FUNCTION_BLOCK FB_System_MVKW_Ablaufsteuerung
VAR_IN_OUT
	Zustand					: ST_System_MVKW_Zustand;
	Stellwert				: ST_System_MVKW_Stellwert;
	Steuerung				: ST_System_MVKW_Steuerung;
END_VAR
VAR_INPUT
	Zustand_Stellventil		: ST_SV_Zustand;
	Zustand_Pumpe			: ST_PU_Zustand;
END_VAR
VAR_OUTPUT
END_VAR
VAR
	E_System_DLK_Zustand_Status_Stoerung	: SINT;
	E_System_DLK_Zustand_Status_Idle_Sperre	: SINT;
END_VAR

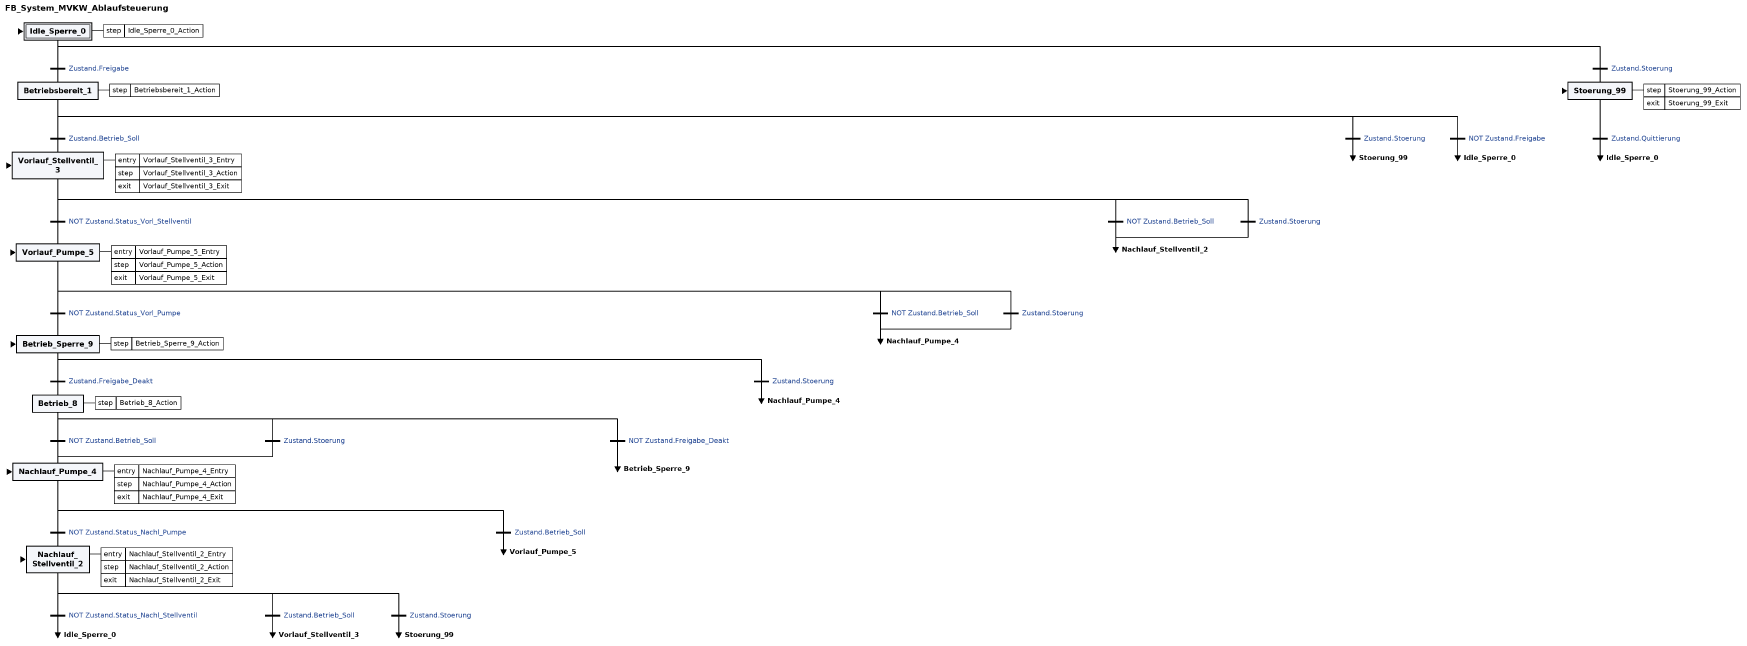
INITIAL_STEP Idle_Sperre_0:
    Idle_Sperre_0_Action(N);  // step action
END_STEP
TRANSITION FROM Idle_Sperre_0 TO Betriebsbereit_1
    := Zustand.Freigabe;
END_TRANSITION
TRANSITION FROM Idle_Sperre_0 TO Stoerung_99
    := Zustand.Stoerung;
END_TRANSITION
STEP Stoerung_99:
    Stoerung_99_Action(N);  // step action
    Stoerung_99_Exit(P0);  // exit action
END_STEP
TRANSITION FROM Stoerung_99 TO Idle_Sperre_0
    := Zustand.Quittierung;
END_TRANSITION
STEP Betriebsbereit_1:
    Betriebsbereit_1_Action(N);  // step action
END_STEP
TRANSITION FROM Betriebsbereit_1 TO Vorlauf_Stellventil_3
    := Zustand.Betrieb_Soll;
END_TRANSITION
TRANSITION FROM Betriebsbereit_1 TO Stoerung_99
    := Zustand.Stoerung;
END_TRANSITION
TRANSITION FROM Betriebsbereit_1 TO Idle_Sperre_0
    := NOT Zustand.Freigabe;
END_TRANSITION
STEP Vorlauf_Stellventil_3:
    Vorlauf_Stellventil_3_Entry(P1);  // entry action
    Vorlauf_Stellventil_3_Action(N);  // step action
    Vorlauf_Stellventil_3_Exit(P0);  // exit action
END_STEP
TRANSITION FROM Vorlauf_Stellventil_3 TO Vorlauf_Pumpe_5
    := NOT Zustand.Status_Vorl_Stellventil;
END_TRANSITION
TRANSITION FROM Vorlauf_Stellventil_3 TO Nachlauf_Stellventil_2
    := NOT Zustand.Betrieb_Soll;
END_TRANSITION
TRANSITION FROM Vorlauf_Stellventil_3 TO Nachlauf_Stellventil_2
    := Zustand.Stoerung;
END_TRANSITION
STEP Vorlauf_Pumpe_5:
    Vorlauf_Pumpe_5_Entry(P1);  // entry action
    Vorlauf_Pumpe_5_Action(N);  // step action
    Vorlauf_Pumpe_5_Exit(P0);  // exit action
END_STEP
TRANSITION FROM Vorlauf_Pumpe_5 TO Betrieb_Sperre_9
    := NOT Zustand.Status_Vorl_Pumpe;
END_TRANSITION
TRANSITION FROM Vorlauf_Pumpe_5 TO Nachlauf_Pumpe_4
    := NOT Zustand.Betrieb_Soll;
END_TRANSITION
TRANSITION FROM Vorlauf_Pumpe_5 TO Nachlauf_Pumpe_4
    := Zustand.Stoerung;
END_TRANSITION
STEP Betrieb_Sperre_9:
    Betrieb_Sperre_9_Action(N);  // step action
END_STEP
TRANSITION FROM Betrieb_Sperre_9 TO Betrieb_8
    := Zustand.Freigabe_Deakt;
END_TRANSITION
TRANSITION FROM Betrieb_Sperre_9 TO Nachlauf_Pumpe_4
    := Zustand.Stoerung;
END_TRANSITION
STEP Betrieb_8:
    Betrieb_8_Action(N);  // step action
END_STEP
TRANSITION FROM Betrieb_8 TO Nachlauf_Pumpe_4
    := NOT Zustand.Betrieb_Soll;
END_TRANSITION
TRANSITION FROM Betrieb_8 TO Nachlauf_Pumpe_4
    := Zustand.Stoerung;
END_TRANSITION
TRANSITION FROM Betrieb_8 TO Betrieb_Sperre_9
    := NOT Zustand.Freigabe_Deakt;
END_TRANSITION
STEP Nachlauf_Pumpe_4:
    Nachlauf_Pumpe_4_Entry(P1);  // entry action
    Nachlauf_Pumpe_4_Action(N);  // step action
    Nachlauf_Pumpe_4_Exit(P0);  // exit action
END_STEP
TRANSITION FROM Nachlauf_Pumpe_4 TO Nachlauf_Stellventil_2
    := NOT Zustand.Status_Nachl_Pumpe;
END_TRANSITION
TRANSITION FROM Nachlauf_Pumpe_4 TO Vorlauf_Pumpe_5
    := Zustand.Betrieb_Soll;
END_TRANSITION
STEP Nachlauf_Stellventil_2:
    Nachlauf_Stellventil_2_Entry(P1);  // entry action
    Nachlauf_Stellventil_2_Action(N);  // step action
    Nachlauf_Stellventil_2_Exit(P0);  // exit action
END_STEP
TRANSITION FROM Nachlauf_Stellventil_2 TO Idle_Sperre_0
    := NOT Zustand.Status_Nachl_Stellventil;
END_TRANSITION
TRANSITION FROM Nachlauf_Stellventil_2 TO Vorlauf_Stellventil_3
    := Zustand.Betrieb_Soll;
END_TRANSITION
TRANSITION FROM Nachlauf_Stellventil_2 TO Stoerung_99
    := Zustand.Stoerung;
END_TRANSITION

ACTION Betrieb_8_Action:
(* Stellwert setzen *)
Stellwert.Anford_Stellventil		:= TRUE;
Stellwert.Anford_Pumpe		:= TRUE;

(* Zustand setzen *)
Zustand.Status				:= E_System_MVKW_Zustand_Status_Betrieb;
END_ACTION

ACTION Betrieb_Sperre_9_Action:
(* Stellwert setzen *)
Stellwert.Anford_Stellventil		:= TRUE;
Stellwert.Anford_Pumpe		:= TRUE;

(* Zustand setzen *)
Zustand.Status				:= E_System_MVKW_Zustand_Status_Betrieb_Sperre;
END_ACTION

ACTION Betriebsbereit_1_Action:
(* Stellwert setzen *)
Stellwert.Anford_Stellventil	:= FALSE;
Stellwert.Anford_Pumpe	:= FALSE;

(* Zustand setzen *)
Zustand.Status			:= E_System_MVKW_Zustand_Status_Betriebsbereit;
END_ACTION

ACTION Idle_Sperre_0_Action:
(* Stellwert setzen *)
Stellwert.Anford_Stellventil	:= FALSE;
Stellwert.Anford_Pumpe	:= FALSE;
Stellwert.Anford_Kompressor		:= FALSE;

(* Zustand setzen *)
Zustand.Status			:= E_System_DLK_Zustand_Status_Idle_Sperre;

(* Quittierungszustand auf False setzen, damit das System bei einer erneuten Störung nicht direkt wieder angeschaltet wird *)
Steuerung.Quittierung	:= FALSE;
END_ACTION

ACTION Nachlauf_Pumpe_4_Action:
(* Stellwert setzen *)
Stellwert.Anford_Stellventil		:= TRUE;
Stellwert.Anford_Pumpe		:= FALSE;

(* Zustand setzen *)
Zustand.Status				:= E_System_MVKW_Zustand_Status_Nachl_Pumpe;
Zustand.Status_Nachl_Pumpe	:= Zustand_Pumpe.Betrieb OR Zustand_Pumpe.Status_Nachl;
END_ACTION

ACTION Nachlauf_Pumpe_4_Entry:
Zustand.Status_Nachl_Pumpe	:= TRUE;
END_ACTION

ACTION Nachlauf_Pumpe_4_Exit:
Zustand.Status_Nachl_Pumpe	:= FALSE;
END_ACTION

ACTION Nachlauf_Stellventil_2_Action:
(* Stellwert setzen *)
Stellwert.Anford_Stellventil		:= FALSE;
Stellwert.Anford_Pumpe		:= FALSE;

(* Zustand setzen *)
Zustand.Status				:= E_System_MVKW_Zustand_Status_Nachl_Stellventil;
Zustand.Status_Nachl_Stellventil	:= Zustand_Stellventil.Stellung OR Zustand_Stellventil.Stellungwechsel10;
END_ACTION

ACTION Nachlauf_Stellventil_2_Entry:
Zustand.Status_Nachl_Stellventil	:= TRUE;
END_ACTION

ACTION Nachlauf_Stellventil_2_Exit:
Zustand.Status_Nachl_Stellventil	:= FALSE;
END_ACTION

ACTION Stoerung_99_Action:
(* Stellwert setzen *)
Stellwert.Anford_Stellventil		:= FALSE;
Stellwert.Anford_Pumpe		:= FALSE;
Stellwert.Anford_Kompressor	:= FALSE;

(* Zustand setzen *)
Zustand.Stoerung			:= TRUE;
Zustand.Status			:= E_System_DLK_Zustand_Status_Stoerung;
END_ACTION

ACTION Stoerung_99_Exit:
Zustand.Stoerung	:= FALSE;
END_ACTION

ACTION Vorlauf_Pumpe_5_Action:
(* Stellwert setzen *)
Stellwert.Anford_Stellventil		:= TRUE;
Stellwert.Anford_Pumpe		:= TRUE;

(* Zustand setzen *)
Zustand.Status				:= E_System_MVKW_Zustand_Status_Vorl_Pumpe;
Zustand.Status_Vorl_Pumpe	:= NOT(Zustand_Pumpe.Betrieb AND NOT Zustand_Pumpe.Status_Vorl);
END_ACTION

ACTION Vorlauf_Pumpe_5_Entry:
Zustand.Status_Vorl_Pumpe	:= TRUE;
END_ACTION

ACTION Vorlauf_Pumpe_5_Exit:
Zustand.Status_Vorl_Pumpe	:= FALSE;
END_ACTION

ACTION Vorlauf_Stellventil_3_Action:
(* Stellwert setzen *)
Stellwert.Anford_Stellventil		:= TRUE;
Stellwert.Anford_Pumpe		:= FALSE;

(* Zustand setzen *)
Zustand.Status				:= E_System_MVKW_Zustand_Status_Vorl_Stellventil;
Zustand.Status_Vorl_Stellventil	:= NOT(Zustand_Stellventil.Stellung AND NOT Zustand_Stellventil.Stellungwechsel01);
END_ACTION

ACTION Vorlauf_Stellventil_3_Entry:
Zustand.Status_Vorl_Stellventil	:= TRUE;
END_ACTION

ACTION Vorlauf_Stellventil_3_Exit:
Zustand.Status_Vorl_Stellventil	:= FALSE;
END_ACTION

END_FUNCTION_BLOCK

(* stored: Version 1.1.0.1, ProductVersion 3.1.4024.9
   POU FB_System_MVKW_Ablaufsteuerung: Id {c04f87bc-0908-44c2-ae40-254fccb8153f}, SpecialFunc None
   Action Betrieb_8_Action: Id {74a05dd1-2be9-4efe-9887-badf43200773}
   Action Betrieb_Sperre_9_Action: Id {caf296c7-fe59-4ff6-8183-9d1c59a55610}
   Action Betriebsbereit_1_Action: Id {76f997f6-180c-49c2-a45f-e541457925d5}
   Action Idle_Sperre_0_Action: Id {806cf063-9d6e-4974-be5c-3aa1ef7ec8b7}
   Action Nachlauf_Pumpe_4_Action: Id {228d89e7-4fbd-445c-9b9d-1960ad6fe3c1}
   Action Nachlauf_Pumpe_4_Entry: Id {bcb9a086-0ff2-4580-b134-d824a4d9f604}
   Action Nachlauf_Pumpe_4_Exit: Id {1181424c-21ff-4ffb-83a2-d01255521d2b}
   Action Nachlauf_Stellventil_2_Action: Id {893289c5-dcc7-4cab-952a-0a0afa6df48f}
   Action Nachlauf_Stellventil_2_Entry: Id {25d54aed-b159-4ab3-84e1-f78cc07f0178}
   Action Nachlauf_Stellventil_2_Exit: Id {283e206e-2676-4bcb-9947-a110b4c4b488}
   Action Stoerung_99_Action: Id {f1369532-5e7a-4b69-90a0-5a681f41a2fa}
   Action Stoerung_99_Exit: Id {3d8f68d8-2370-4aae-8777-2d5bec9c6c43}
   Action Vorlauf_Pumpe_5_Action: Id {8bdb9eed-9af4-4eb2-9f13-6a2200b98d85}
   Action Vorlauf_Pumpe_5_Entry: Id {dc07c885-c8b1-486a-a015-ffb5b94dab16}
   Action Vorlauf_Pumpe_5_Exit: Id {d40f7cbd-f382-40cf-a3e7-dfae894db278}
   Action Vorlauf_Stellventil_3_Action: Id {0614c1a9-9925-44ec-a7f6-9f2878c5512a}
   Action Vorlauf_Stellventil_3_Entry: Id {d0dd7ee8-6276-46cf-9f10-6eb10636e699}
   Action Vorlauf_Stellventil_3_Exit: Id {702e9a57-0135-4a4c-9262-8ed84836b165} *)
